// TIA Portal V19 export
DATA_BLOCK "1200Comm_DB"   // DB2
// stored: InstanceOfName 1200Comm, InstanceOfType FB
"1200Comm"
BEGIN
END_DATA_BLOCK
